RoboDK station: Stitching with sticher using Fanuc.rdk

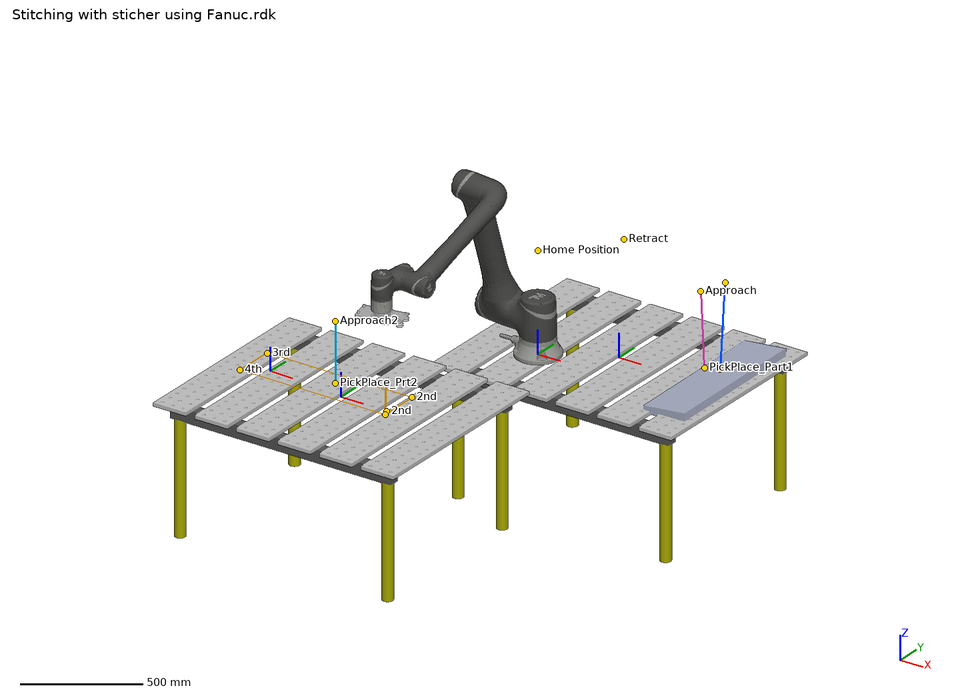
[picture v0: the station drawn from its stored meshes, robots at their saved joint values, targets as dots, program paths as lines]
Station Stitching with sticher using Fanuc (saved by RoboDK 5.1.0). Poses are relative to the parent item; angles as X-Y-Z fixed-axis rotations.
Station parameters (name, value as stored): OPC-UA, opc.tcp://localhost:4840
  - frame Frame 2 at (-849.61, -404.11, 112.6) mm
    - target Home Position (Cartesian target) at (550.89, 609.76, 573.04) mm, rotated rx -178.84 ry 60.9 rz -179.86 deg; joints [-18.502, -38.59, 118.247, -49.418, 105.073, -99.264] of Omron TM12X
    - target Retract (Cartesian target) at (930.89, 679.76, 703.04) mm, rotated rx -173.84 ry 45.9 rz -174.86 deg; joints [2.137, -2.643, 73.991, -27.43, 86, -92.092] of Omron TM12X
    - target Approach (Cartesian target) at (924.81, 1233.71, 243.56) mm, rotated rx 179.4 ry 2.27 rz -178.66 deg; joints [36.144, 26.738, 88.534, -27.482, 89.197, -145.226] of Omron TM12X
    - target PickPlace_Part1 (Cartesian target) at (940.37, 1235.87, -99.57) mm, rotated rx -179.05 ry -0.07 rz -178.55 deg; joints [35.67, 47.381, 94.458, -51.245, 89.251, -145.772] of Omron TM12X
    - object Table at (0, 0, 0) mm, size 1193.8 x 965.2 x 609.6 mm, geometry from welding_table.sld
      - object 197143A at (880.42, 891.33, -183.84) mm, rotated rx 174.92 ry 0.04 rz 90.81 deg, size 734 x 204 x 35 mm, geometry from 197143A.IGS
  - frame Object at (-329.47, 825.84, -55.54) mm
    - object Table at (0, 0, 0) mm, size 1193.8 x 965.2 x 609.6 mm, geometry from welding_table.sld
  - frame Drop at (-1209.15, -394.59, 123.51) mm
    - target Approach2 (Cartesian target) at (319.83, 8.55, 311.87) mm, rotated rx -178.81 ry -0.1 rz 92.19 deg; joints [-88.823, 16.471, 94.157, -20.547, 88.807, -181.01]
    - target PickPlace_Prt2 (Cartesian target) at (319.83, 8.55, 31.87) mm, rotated rx -178.81 ry -0.1 rz 92.19 deg; joints [-88.823, 30.903, 106.753, -47.575, 88.807, -181.01]
  - program ReplaceObjects (1 instructions, listed below)
  - program PickPart1 (6 instructions, listed below)
  - program PlacePart2 (6 instructions, listed below)
  - program PickPart2 (6 instructions, listed below)
  - program MainProgram (4 instructions, listed below)
  - program PlacePart1 (6 instructions, listed below)
  - frame Frame 8 at (0, 2825.84, 0) mm
  - frame Frame 7 at (0, 3825.84, 0) mm
    - target 2nd (Cartesian target) at (-575.97, -4297.87, 150.37) mm, rotated rx -180 ry 0 rz 0 deg; joints [-3.584, 106.943, 80, 103.359]
    - target Apr1 (Cartesian target) at (-575.97, -4297.87, 280.37) mm, rotated rx -180 ry 0 rz 0 deg; joints [-3.584, 106.943, 210, 103.359]
    - target 1st (Cartesian target) at (-575.97, -4307.87, 140.37) mm, rotated rx -180 ry 0 rz 0 deg; joints [-5.257, 108.461, 70, 103.205]
    - target 2nd (Cartesian target) at (-575.97, -4117.87, 140.37) mm, rotated rx -180 ry 0 rz 0 deg; joints [25.754, 70.991, 70, 96.745]
    - target 3rd (Cartesian target) at (-1295.97, -4117.87, 140.37) mm, rotated rx -180 ry 0 rz 0 deg; joints [120.978, 29.039, 70, 150.017]
    - target 4th (Cartesian target) at (-1295.97, -4307.87, 140.37) mm, rotated rx -180 ry 0 rz 0 deg; joints [114.601, 76.591, 70, 191.192]
    - target 5th (Cartesian target) at (-575.97, -4307.87, 140.37) mm, rotated rx -180 ry 0 rz 0 deg; joints [-5.257, 108.461, 70, 103.205]
  - program Prog7 (8 instructions, listed below)
  - frame Omron TM12X Base at (-552.68, 569.71, 0) mm
    - robot Omron TM12X: 6 axes, payload 12 kg, reach 1300 mm, repeatability 0.1 mm, weight 33.3 kg
        modified DH rows (alpha deg, a mm, theta deg, d mm): 0, 0, 0, 165.2; 90, 0, 90, 0; 0, 636.1, 0, 0; 0, 557.9, -90, 156.3; -90, 0, 0, 106; 90, 0, 180, 113.15
        joint limits [-270, -180, -166, -180, -180, -270] to [270, 180, 166, 180, 180, 270]; home [0, 0, 90, 0, 90, 0]; saved at [-94.1, 17.51, 93.897, -21.641, 89.243, -197.42]
      - tool GripperA, TCP at (0, 0, 30) mm, rotated rx 0 ry 0 rz 90 deg, size 209.9 x 42 x 100 mm
  - frame Frame 8 at (0, 4825.84, 0) mm
    - target Appr. (Cartesian target) at (-889.32, -5211.87, 435.38) mm, rotated rx -178.81 ry -0.1 rz 92.19 deg; joints [-100.361, 33.294, 68.989, -12.442, 88.815, -192.55] of Omron TM12X
    - target Pick. (Cartesian target) at (-889.32, -5211.87, 155.38) mm, rotated rx -178.81 ry -0.1 rz 92.19 deg; joints [-100.361, 43.901, 81.771, -35.83, 88.815, -192.55] of Omron TM12X
  - program Prog8 (5 instructions, listed below)
  - frame Frame 9 at (0, 5825.84, 0) mm
    - target Appro1 (Cartesian target) at (109.28, -4873.24, 355.39) mm, rotated rx -178.8 ry 4.9 rz -176.81 deg; joints [-33.359, 25.69, 90.822, -31.162, 91.95, -216.423] of Omron TM12X
    - target Drop (Cartesian target) at (119.28, -4923.24, -14.61) mm, rotated rx -178.8 ry 4.9 rz -176.81 deg; joints [-35.617, 50.365, 93.649, -58.584, 92.132, -218.675] of Omron TM12X
  - program Prog9 (5 instructions, listed below)
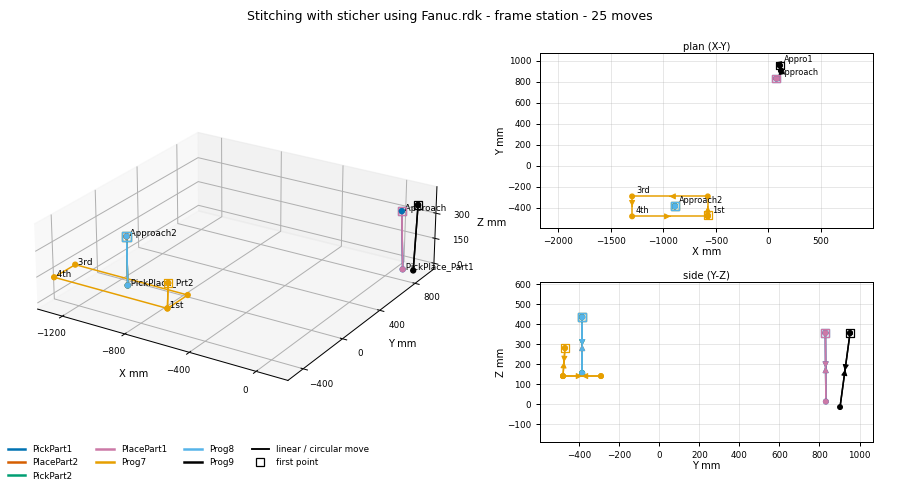
[picture p0: tool path of Stitching with sticher using Fanuc.rdk in frame station, 25 of 25 moves have a stored position in this frame; points joined in program order, loops and branches not executed]

--- program ReplaceObjects (robot Omron TM12X) ---
  Replace objects

--- program PickPart1 (robot Omron TM12X) ---
  Set Ref.: Frame 2
  Set Tool: GripperA at (0, 0, 30) mm, rotated rx 0 ry 0 rz 90 deg
  MoveJ (Approach)
  MoveL (PickPlace_Part1)
  Attach to GripperA
  MoveL (Approach)

--- program PlacePart2 (robot Omron TM12X) ---
  Set Ref.: Drop
  Set Tool: GripperA at (0, 0, 30) mm, rotated rx 0 ry 0 rz 90 deg
  MoveJ (Approach2)
  MoveL (PickPlace_Prt2)
  Detach from GripperA
  MoveL (Approach2)

--- program PickPart2 (robot Omron TM12X) ---
  Set Ref.: Drop
  Set Tool: GripperA at (0, 0, 30) mm, rotated rx 0 ry 0 rz 90 deg
  MoveJ (Approach2)
  MoveL (PickPlace_Prt2)
  Attach to GripperA
  MoveL (PickPlace_Prt2)

--- program MainProgram (robot Omron TM12X) ---
  Call PickPart1
  Call PlacePart2
  Call PickPart2
  Call PlacePart1

--- program PlacePart1 (robot Omron TM12X) ---
  Set Ref.: Frame 2
  Set Tool: GripperA at (0, 0, 30) mm, rotated rx 0 ry 0 rz 90 deg
  MoveJ (Approach)
  MoveL (PickPlace_Part1)
  Detach from GripperA
  MoveL (Approach)

--- program Prog7 ---
  Set Ref.: Frame 7
  MoveL (Apr1)
  MoveL (1st)
  MoveL (2nd)
  MoveL (3rd)
  MoveL (4th)
  MoveL (5th)
  MoveL (Apr1)

--- program Prog8 (robot Omron TM12X) ---
  Set Ref.: Frame 8
  MoveL (Appr.)
  MoveL (Pick.)
  Attach to GripperA
  MoveL (Appr.)

--- program Prog9 (robot Omron TM12X) ---
  Set Ref.: Frame 9
  MoveL (Appro1)
  MoveL (Drop)
  Detach from GripperA
  MoveL (Appro1)
